TYPE ST_ResidualCurrentMonitor_get :
STRUCT
	b_prewarning			: BOOL;
END_STRUCT
END_TYPE

(* stored: Version 1.1.0.1, ProductVersion 3.1.4024.12
   DUT ST_ResidualCurrentMonitor_get: Id {b15443d4-2595-4749-9ec6-01f7d7316fe7} *)
